{attribute 'qualified_only'}
VAR_GLOBAL
	

saydir1: TON;
start:BOOL;
cikis:BOOL;
gecensure:TIME;
gecenzaman:INT;
hesaplama:INT;






END_VAR

(* stored: Version 1.1.0.1, ProductVersion 3.1.4024.12
   GVL GVL_hesapSayfa: Id {52eaa716-6ffe-4a01-8201-f9ad22cdb3b3} *)
